% RSLogix 500 project CLOCK.RSS, saved by version 8.30.00.16 %
PROJECT "UNTITLED"    % processor: MicroLogix 1000 %

PROGRAM FILES
  LAD 2 "MAIN_PROG"  18 rungs
  LAD 3 "USER_FAULT"  1 rungs
  LAD 4 "HSC_INT"  1 rungs
  LAD 5 "STI_INT"  1 rungs
  LAD 6, 7, 8, 9, 10, 11, 12, 13, 14, 15, 16: only END

DATA FILES
  O0 OUTPUT  1 elements
  I1 INPUT  2 elements
  S2 STATUS  33 elements
  B3 BINARY  32 elements
  T4 TIMER  40 elements
  C5 COUNTER  32 elements
  R6 CONTROL  16 elements
  N7 INTEGER  105 elements

LADDER 2 "MAIN_PROG"
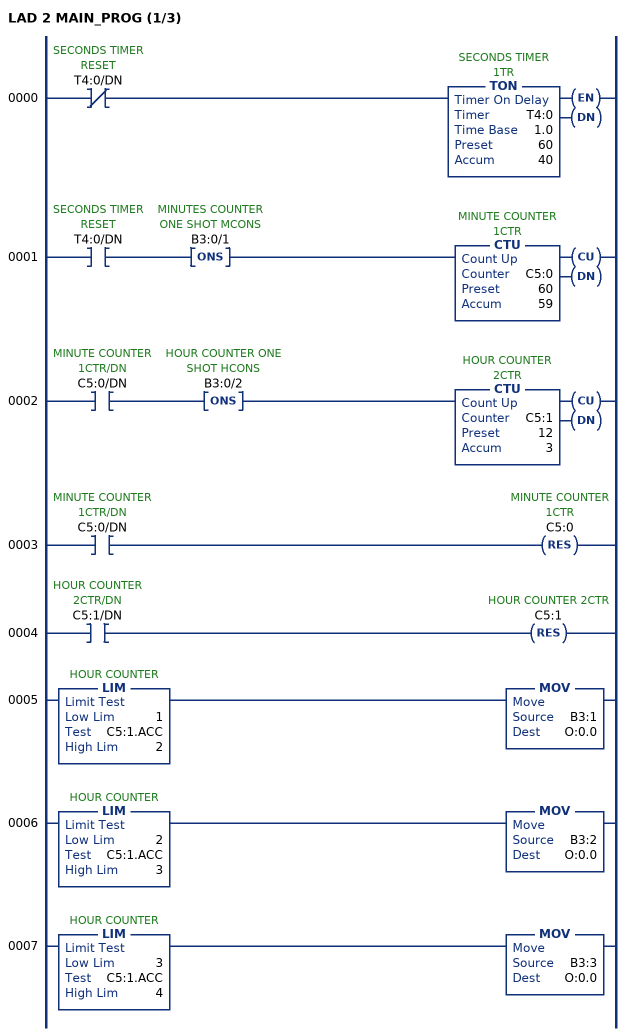
% Rung: 0 %
SOR XIO T4:0/DN TON T4:0 1.0 60 40 EOR
%   T4:0/DN  "SECONDS TIMER RESET" %
%   T4:0  1TR  "SECONDS TIMER" %
% Rung: 1 %
SOR XIC T4:0/DN OSR B3:0/1 CTU C5:0 60 59 EOR
%   T4:0/DN  "SECONDS TIMER RESET" %
%   B3:0/1  MCONS  "MINUTES COUNTER ONE SHOT" %
%   C5:0  1CTR  "MINUTE COUNTER" %
% Rung: 2 %
SOR XIC C5:0/DN OSR B3:0/2 CTU C5:1 12 3 EOR
%   C5:0  1CTR  "MINUTE COUNTER" %
%   B3:0/2  HCONS  "HOUR COUNTER ONE SHOT" %
%   C5:1  2CTR  "HOUR COUNTER" %
% Rung: 3 %
SOR XIC C5:0/DN RES C5:0 EOR
%   C5:0  1CTR  "MINUTE COUNTER" %
% Rung: 4 %
SOR XIC C5:1/DN RES C5:1 EOR
%   C5:1  2CTR  "HOUR COUNTER" %
% Rung: 5 %
SOR LIM 1 C5:1.ACC 2 MOV B3:1 O:0.0 EOR
%   C5:1.ACC  "HOUR COUNTER" %
% Rung: 6 %
SOR LIM 2 C5:1.ACC 3 MOV B3:2 O:0.0 EOR
%   C5:1.ACC  "HOUR COUNTER" %
% Rung: 7 %
SOR LIM 3 C5:1.ACC 4 MOV B3:3 O:0.0 EOR
%   C5:1.ACC  "HOUR COUNTER" %

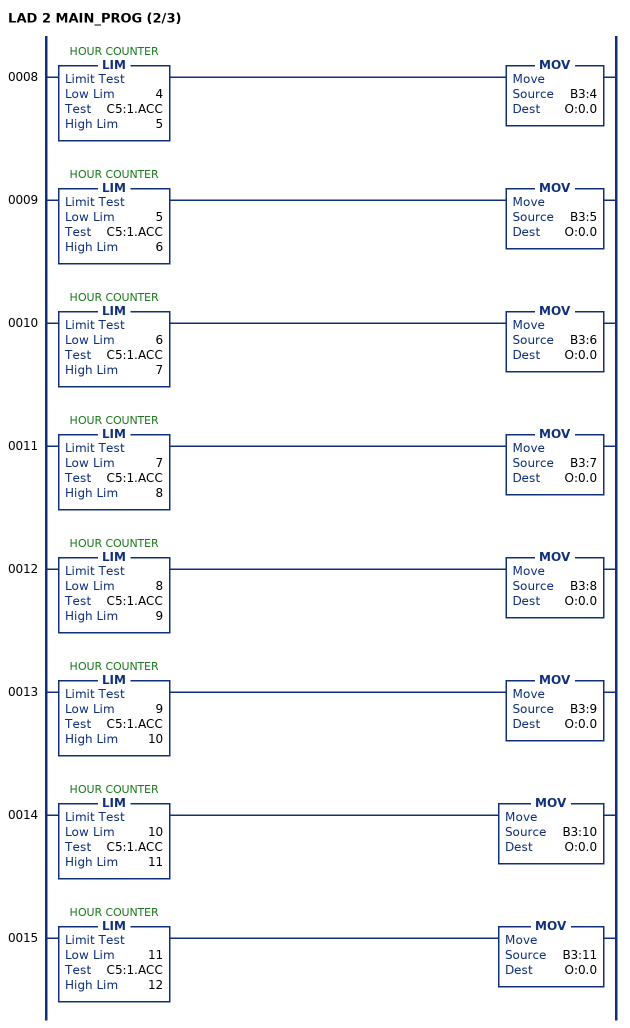
% Rung: 8 %
SOR LIM 4 C5:1.ACC 5 MOV B3:4 O:0.0 EOR
%   C5:1.ACC  "HOUR COUNTER" %
% Rung: 9 %
SOR LIM 5 C5:1.ACC 6 MOV B3:5 O:0.0 EOR
%   C5:1.ACC  "HOUR COUNTER" %
% Rung: 10 %
SOR LIM 6 C5:1.ACC 7 MOV B3:6 O:0.0 EOR
%   C5:1.ACC  "HOUR COUNTER" %
% Rung: 11 %
SOR LIM 7 C5:1.ACC 8 MOV B3:7 O:0.0 EOR
%   C5:1.ACC  "HOUR COUNTER" %
% Rung: 12 %
SOR LIM 8 C5:1.ACC 9 MOV B3:8 O:0.0 EOR
%   C5:1.ACC  "HOUR COUNTER" %
% Rung: 13 %
SOR LIM 9 C5:1.ACC 10 MOV B3:9 O:0.0 EOR
%   C5:1.ACC  "HOUR COUNTER" %
% Rung: 14 %
SOR LIM 10 C5:1.ACC 11 MOV B3:10 O:0.0 EOR
%   C5:1.ACC  "HOUR COUNTER" %
% Rung: 15 %
SOR LIM 11 C5:1.ACC 12 MOV B3:11 O:0.0 EOR
%   C5:1.ACC  "HOUR COUNTER" %

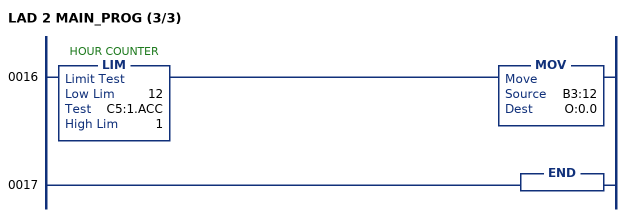
% Rung: 16 %
SOR LIM 12 C5:1.ACC 1 MOV B3:12 O:0.0 EOR
%   C5:1.ACC  "HOUR COUNTER" %
% Rung: 17 %
SOR END EOR

OTHER DOCUMENTED ADDRESSES
  B3:0/0  SSP  "SPRINKLER START PERMISSIVE"
  B3:0/3  "SPRINKLER SYSTEM START PERMISSIVE"
  B3:0/4  STCP  "SPRINKLER TIMER SYSLE PERMISSIVE"
  I:0.0/0  1PB  "SPRIKLER STOP"
  I:0.0/1  2PB  "SPRINKLER CLOCK MANUAL START"
  O:0.0/0  1SV  "SPRINKLER VALVE 1"
  O:0.0/1  2SV  "SPRINKLER VALVE 2"
  O:0.0/2  3SV  "SPRINKLER VALVE 3"
  O:0.0/3  4SV  "SPRINKLER VALVE 4"
  T4:1  1SVT  "SPRINKLER VALVE 1 TIMER"
  T4:2  2SVT  "SPRINKLER VALVE 2 TIMER"
  T4:3  3SVT  "SPRINKLER VALVE 3 TIMER"
  T4:4  4SVT  "SPRINKLER VALVE 4 TIMER"

DATA TABLE (non-zero values as saved)
DATA B3
% B3:0 % 0X0000 0X0001 0X0002 0X0003 0X0004 0X0005 0X0006 0X0007 0X0008 0X0009
% B3:10 % 0X000A 0X000B 0X000C 0X000D 0X000E 0X000F 0X000F 0X0000 0X0000 0X0000
DATA T4
% .PRE .ACC %
% T4:0 % 60 40
% T4:1 % 10 0
% T4:2 % 10 0
% T4:3 % 10 0
% T4:4 % 10 0
DATA C5
% .PRE .ACC %
% C5:0 % 60 59
% C5:1 % 12 3
